// TIA Portal V19 export
FUNCTION "FC_Niveau_St" : Void   // FC96, STL
TITLE = Badniveau-Steuerungen
{ S7_Optimized_Access := 'FALSE' }
AUTHOR : RE
NAME : FC_nass
VERSION : 2.0
// stored: AutoNumber false
   VAR_TEMP
      Freigabe : Bool;
   END_VAR
BEGIN

NETWORK
TITLE = Niveau-Regelungen/Nachspeisungen/Spritzregister
      CLR;
      =     "DB_NSP".Test_on;

      CALL  "FC_Nachspeisung";

      A     "DB_ANLAGE".BA.Simulation;
      BEC;


NETWORK
TITLE = CM01
      A     "Panel".CM01.NSP_Auto;
      =     "DB_Panel_Posinfo".Pos[1].NS_Auto;

// Becken leer und keine Dosierung aktiv
      AN    "DB_POS".POS[1].belegt;
      AN    "DB_POS".POS[2].belegt;
      AN    "DB_POS".POS[3].belegt;
      AN    "DB_POS".POS[4].belegt;
      AN    "DB_POS".POS[5].belegt;
      AN    "DB_POS".POS[6].belegt;
      AN    "DB_DP".DP[1].Dosi_akt;
      AN    "DB_DP".DP[2].Dosi_akt;
      AN    "DB_DP".DP[5].Dosi_akt;
      AN    "DB_DP".DP[6].Dosi_akt;
      =     "DB_NSP".NSP[1].Freigabe;

      A     "E_Niv_Min_CM01.BL03";
      =     "DB_NSP".NSP[1].Niveau_ok;
      =     "DB_NSP".NSP[2].Niveau_ok;
      =     "DB_NSP".NSP[3].Niveau_ok;
      =     "DB_NSP".NSP[4].Niveau_ok;
      =     "DB_NSP".NSP[5].Niveau_ok;
      =     "DB_NSP".NSP[6].Niveau_ok;
      NOT;
      =     "DB_NSP".NSP[1].AL_Niv_min;

// Dosierungen gegeneinander verriegeln
// Verwerfen hat Vorrang
      A     "DB_DP".DP[1].Dosi_akt;
      O     "DB_DP".DP[5].Dosi_akt;
      O     "DB_DP".DP[3].Dosi_akt;
      O     "DB_DP".DP[7].Dosi_akt;
      S     "DB_DP".DP[2].DP_OFF;
      S     "DB_DP".DP[6].DP_OFF;
      S     "DB_DP".DP[4].DP_OFF;
      S     "DB_DP".DP[8].DP_OFF;
      JC    Ents;

// CM01 gewinnt
      A     "DB_DP".DP[2].Dosi_akt;  //CM01
      O     "DB_DP".DP[6].Dosi_akt;
      A(;
      A     "DB_DP".DP[4].Dosi_akt;  //CM02
      O     "DB_DP".DP[8].Dosi_akt;
      );
      AN    "DB_DP".DP[2].DP_OFF;
      AN    "DB_DP".DP[6].DP_OFF;
      S     "DB_DP".DP[4].DP_OFF;
      S     "DB_DP".DP[8].DP_OFF;
      JC    Ents;

      A     "DB_DP".DP[2].Dosi_akt;  //CM01
      O     "DB_DP".DP[6].Dosi_akt;
      AN    "DB_DP".DP[2].DP_OFF;
      AN    "DB_DP".DP[6].DP_OFF;
      =     "DB_DP".DP[4].DP_OFF;
      =     "DB_DP".DP[8].DP_OFF;

      A     "DB_DP".DP[4].Dosi_akt;  //CM02
      O     "DB_DP".DP[8].Dosi_akt;
      AN    "DB_DP".DP[4].DP_OFF;
      AN    "DB_DP".DP[8].DP_OFF;
      =     "DB_DP".DP[2].DP_OFF;
      =     "DB_DP".DP[6].DP_OFF;

//Verwerfen - alles aus
Ents: AN    "DB_DP".DP[1].Dosi_akt;
      AN    "DB_DP".DP[3].Dosi_akt;
      AN    "DB_DP".DP[5].Dosi_akt;
      AN    "DB_DP".DP[7].Dosi_akt;
      R     "DB_DP".DP[1].DP_OFF;
      R     "DB_DP".DP[3].DP_OFF;
      R     "DB_DP".DP[5].DP_OFF;
      R     "DB_DP".DP[7].DP_OFF;

// Verwerfen CM01 gewinnt
      A     "DB_DP".DP[1].Dosi_akt;  //CM01
      O     "DB_DP".DP[5].Dosi_akt;
      A(;
      A     "DB_DP".DP[3].Dosi_akt;  //CM02
      O     "DB_DP".DP[7].Dosi_akt;
      );
      AN    "DB_DP".DP[1].DP_OFF;
      AN    "DB_DP".DP[5].DP_OFF;
      S     "DB_DP".DP[3].DP_OFF;
      S     "DB_DP".DP[7].DP_OFF;
      JC    CM01;

      A     "DB_DP".DP[1].Dosi_akt;  //CM01
      O     "DB_DP".DP[5].Dosi_akt;
      AN    "DB_DP".DP[1].DP_OFF;
      AN    "DB_DP".DP[5].DP_OFF;
      =     "DB_DP".DP[3].DP_OFF;
      =     "DB_DP".DP[7].DP_OFF;

      A     "DB_DP".DP[3].Dosi_akt;  //CM02
      O     "DB_DP".DP[7].Dosi_akt;
      AN    "DB_DP".DP[3].DP_OFF;
      AN    "DB_DP".DP[7].DP_OFF;
      =     "DB_DP".DP[1].DP_OFF;
      =     "DB_DP".DP[5].DP_OFF;

CM01: NOP   0;
// Anforderung bilden
// Nachschärfen
      A     "DB_NSP".NSP[1].Nachspeisen;
      O(;
      A     "DB_DP".DP[2].Dosi_akt;
      AN    "DB_DP".DP[2].DP_OFF;
      );
      O(;
      A     "DB_DP".DP[6].Dosi_akt;
      AN    "DB_DP".DP[6].DP_OFF;
      );
      A     "Pu_GP01.GP13".In.Auto;
      A     "Pu_GP01.GP13".Out.Versorgung_UV01;
      AN    "Pu_GP02.GP10".In.Anf_HF_CM01;
      =     "Pu_GP01.GP13".In.Anf_HF_CM01;

      A     "DB_NSP".NSP[1].Nachspeisen;
      O(;
      A     "DB_DP".DP[2].Dosi_akt;
      AN    "DB_DP".DP[2].DP_OFF;
      );
      O(;
      A     "DB_DP".DP[6].Dosi_akt;
      AN    "DB_DP".DP[6].DP_OFF;
      );
      A     "Pu_GP02.GP10".In.Auto;
      A     "Pu_GP02.GP10".Out.Versorgung_UV01;
      AN    "Pu_GP01.GP13".In.Anf_HF_CM01;
      =     "Pu_GP02.GP10".In.Anf_HF_CM01;

// Verwerfen
      A     "DB_DP".DP[1].Dosi_akt;
      AN    "DB_DP".DP[1].DP_OFF;
      O(;
      A     "DB_DP".DP[5].Dosi_akt;
      AN    "DB_DP".DP[5].DP_OFF;
      );
      A     "UP_CM01.GP02".In.Auto;
      A(;
      A     "UP_CM01.GP02".In."SRM_GP01.QM14_auf";
      O     "UP_CM01.GP02".In."SRM_GP02.QM41_auf";
      );
      =     "UP_CM01.GP02".In.Anf_HF_Ents_CM0x;

// WT-zählergesteuert (DP1/2)
      A     "Panel".CM01.Dosierung_LF;
      R     "DB_Panel_DP".DoPu[1].Auto;
      R     "DB_Panel_DP".DoPu[2].Auto;

// LF-gesteuert (DP(5/6)
      CALL  "ToDo";

      A     "DB_DP".DP[5].Dosi_akt;
      O     "DB_DP".DP[6].Dosi_akt;
      L     S5T#15m;
      SF    "TA-Pause_LF_CM01";

      AN    "Panel".CM01.Dosierung_LF;
      R     "DB_Panel_DP".DoPu[5].Auto;
      R     "DB_Panel_DP".DoPu[6].Auto;
      JC    LF1E;

      L     "Panel".IW."LF_CM01.BN02";
      L     "Panel".CM01.Sollwert_LF;
      <R;  // ???
      AN    "TA-Pause_LF_CM01";
      AN    "DB_DP".DP[5].AM_DP_Start;
      AN    "DB_DP".DP[6].AM_DP_Start;
      S     "DB_DP".DP[5].DP_Start;
      S     "DB_DP".DP[5].AM_DP_Start;
      S     "DB_DP".DP[6].DP_Start;
      S     "DB_DP".DP[6].AM_DP_Start;
      JC    LF1E;

      A     "DB_DP".DP[5].Dosi_akt;
      R     "DB_DP".DP[5].AM_DP_Start;

      A     "DB_DP".DP[6].Dosi_akt;
      R     "DB_DP".DP[6].AM_DP_Start;

LF1E: NOP   0;


NETWORK
TITLE = CM02
      A     "Panel".CM02.NSP_Auto;
      =     "DB_Panel_Posinfo".Pos[13].NS_Auto;

// Becken leer und keine Dosierung aktiv
      AN    "DB_POS".POS[13].belegt;
      AN    "DB_POS".POS[14].belegt;
      AN    "DB_POS".POS[15].belegt;
      AN    "DB_POS".POS[16].belegt;
      AN    "DB_POS".POS[17].belegt;
      AN    "DB_POS".POS[18].belegt;
      AN    "DB_DP".DP[3].Dosi_akt;
      AN    "DB_DP".DP[4].Dosi_akt;
      AN    "DB_DP".DP[7].Dosi_akt;
      AN    "DB_DP".DP[8].Dosi_akt;
      =     "DB_NSP".NSP[13].Freigabe;

      A     "E_Niv_Min_CM02.BL10";
      =     "DB_NSP".NSP[13].Niveau_ok;
      =     "DB_NSP".NSP[14].Niveau_ok;
      =     "DB_NSP".NSP[15].Niveau_ok;
      =     "DB_NSP".NSP[16].Niveau_ok;
      =     "DB_NSP".NSP[17].Niveau_ok;
      =     "DB_NSP".NSP[18].Niveau_ok;
      NOT;
      =     "DB_NSP".NSP[13].AL_Niv_min;


// Anforderung bilden
// Nachschärfen
      A     "DB_NSP".NSP[13].Nachspeisen;
      O(;
      A     "DB_DP".DP[4].Dosi_akt;
      AN    "DB_DP".DP[4].DP_OFF;
      );
      O(;
      A     "DB_DP".DP[8].Dosi_akt;
      AN    "DB_DP".DP[8].DP_OFF;
      );
      A     "Pu_GP01.GP13".In.Auto;
      A     "Pu_GP01.GP13".Out.Versorgung_UV01;
      AN    "Pu_GP02.GP10".In.Anf_HF_CM02;
      =     "Pu_GP01.GP13".In.Anf_HF_CM02;

      A     "DB_NSP".NSP[13].Nachspeisen;
      O(;
      A     "DB_DP".DP[4].Dosi_akt;
      AN    "DB_DP".DP[4].DP_OFF;
      );
      O(;
      A     "DB_DP".DP[8].Dosi_akt;
      AN    "DB_DP".DP[8].DP_OFF;
      );
      A     "Pu_GP02.GP10".In.Auto;
      A     "Pu_GP02.GP10".Out.Versorgung_UV01;
      AN    "Pu_GP01.GP13".In.Anf_HF_CM02;
      =     "Pu_GP02.GP10".In.Anf_HF_CM02;

// Verwerfen
      A     "DB_DP".DP[3].Dosi_akt;
      AN    "DB_DP".DP[3].DP_OFF;
      O(;
      A     "DB_DP".DP[7].Dosi_akt;
      AN    "DB_DP".DP[7].DP_OFF;
      );
      A     "UP_CM02.GP05".In.Auto;
      A(;
      A     "UP_CM02.GP05".In."SRM_GP01.QM14_auf";
      O     "UP_CM02.GP05".In."SRM_GP02.QM41_auf";
      );
      =     "UP_CM02.GP05".In.Anf_HF_Ents_CM0x;

// WT-zählergesteuert (DP3/4)
      A     "Panel".CM02.Dosierung_LF;
      R     "DB_Panel_DP".DoPu[3].Auto;
      R     "DB_Panel_DP".DoPu[4].Auto;

// LF-gesteuert (DP(7/8)
      CALL  "ToDo";

      A     "DB_DP".DP[7].Dosi_akt;
      O     "DB_DP".DP[8].Dosi_akt;
      L     S5T#15m;
      SF    "TA-Pause_LF_CM02";

      AN    "Panel".CM02.Dosierung_LF;
      R     "DB_Panel_DP".DoPu[7].Auto;
      R     "DB_Panel_DP".DoPu[8].Auto;
      JC    LF2E;

      L     "Panel".IW."LF_CM02.BN04";
      L     "Panel".CM02.Sollwert_LF;
      <R;  // ???
      AN    "TA-Pause_LF_CM02";
      AN    "DB_DP".DP[7].AM_DP_Start;
      AN    "DB_DP".DP[8].AM_DP_Start;
      S     "DB_DP".DP[7].DP_Start;
      S     "DB_DP".DP[7].AM_DP_Start;
      S     "DB_DP".DP[8].DP_Start;
      S     "DB_DP".DP[8].AM_DP_Start;
      JC    LF2E;

      A     "DB_DP".DP[7].Dosi_akt;
      R     "DB_DP".DP[7].AM_DP_Start;

      A     "DB_DP".DP[8].Dosi_akt;
      R     "DB_DP".DP[8].AM_DP_Start;

LF2E: NOP   0;


NETWORK
TITLE = CM03

      A     "Panel".CM03.SPR_Auto;
      =     "DB_Panel_Posinfo".Pos[7].SR_Auto;
      =     "DB_Panel_Posinfo".Pos[8].SR_Auto;
      =     "DB_Panel_Posinfo".Pos[9].SR_Auto;
      =     "DB_Panel_Posinfo".Pos[10].SR_Auto;
      =     "DB_Panel_Posinfo".Pos[11].SR_Auto;
      =     "DB_Panel_Posinfo".Pos[12].SR_Auto;

      A     "Panel".CM03.SPR_Start_Test;
      R     "Panel".CM03.SPR_Start_Test;
      JCN   ST03;
      L     "Panel".CM03.SPR_Zeit_Test;
      T     "DB_Panel_Posinfo".Pos[7].T_Zt_SR;

ST03: A     "Panel".CM03.SPR_Stopp_Test;
      R     "Panel".CM03.SPR_Stopp_Test;
      JCN   FN03;
      L     0;
      T     "DB_Panel_Posinfo".Pos[7].T_Zt_SR;

//Pos.7..12
FN03: AN    "T_VEW_niO";
      A     "E_Niv_Uel_CM05.BL12";
      =     "DB_NSP".NSP[7].Freigabe;
      =     "DB_NSP".NSP[8].Freigabe;
      =     "DB_NSP".NSP[9].Freigabe;
      =     "DB_NSP".NSP[10].Freigabe;
      =     "DB_NSP".NSP[11].Freigabe;
      =     "DB_NSP".NSP[12].Freigabe;

// Spritzregister: beim Heben und Senken
      A     "DB_NSP".NSP[7].Spritzen;
      O     "DB_NSP".NSP[8].Spritzen;
      O     "DB_NSP".NSP[9].Spritzen;
      O     "DB_NSP".NSP[10].Spritzen;
      O     "DB_NSP".NSP[11].Spritzen;
      O     "DB_NSP".NSP[12].Spritzen;
      AN    "T_VEW_niO";
      A     "E_Niv_Uel_CM05.BL12";
      =     "A_CM03.QM35";


NETWORK
TITLE = CM04
//Pos.19..24
      A     "Panel".CM04.SPR_Auto;
      =     "DB_Panel_Posinfo".Pos[19].SR_Auto;
      =     "DB_Panel_Posinfo".Pos[20].SR_Auto;
      =     "DB_Panel_Posinfo".Pos[21].SR_Auto;
      =     "DB_Panel_Posinfo".Pos[22].SR_Auto;
      =     "DB_Panel_Posinfo".Pos[23].SR_Auto;
      =     "DB_Panel_Posinfo".Pos[24].SR_Auto;

      A     "Panel".CM04.NSP_Auto;
      =     "DB_Panel_Posinfo".Pos[19].NS_Auto;
      =     "DB_Panel_Posinfo".Pos[20].NS_Auto;
      =     "DB_Panel_Posinfo".Pos[21].NS_Auto;
      =     "DB_Panel_Posinfo".Pos[22].NS_Auto;
      =     "DB_Panel_Posinfo".Pos[23].NS_Auto;
      =     "DB_Panel_Posinfo".Pos[24].NS_Auto;

      L     "Panel".CM04.NSP_Zeit;
      T     "DB_Panel_Posinfo".Pos[19].Zeit_NS;
      T     "DB_Panel_Posinfo".Pos[20].Zeit_NS;
      T     "DB_Panel_Posinfo".Pos[21].Zeit_NS;
      T     "DB_Panel_Posinfo".Pos[22].Zeit_NS;
      T     "DB_Panel_Posinfo".Pos[23].Zeit_NS;
      T     "DB_Panel_Posinfo".Pos[24].Zeit_NS;

      A     "Panel".CM04.SPR_Start_Test;
      R     "Panel".CM04.SPR_Start_Test;
      JCN   ST04;
      L     "Panel".CM04.SPR_Zeit_Test;
      T     "DB_Panel_Posinfo".Pos[19].T_Zt_SR;

ST04: A     "Panel".CM04.SPR_Stopp_Test;
      R     "Panel".CM04.SPR_Stopp_Test;
      JCN   NS04;
      L     0;
      T     "DB_Panel_Posinfo".Pos[19].T_Zt_SR;

NS04: A     "Panel".CM04.NSP_Start_Test;
      R     "Panel".CM04.NSP_Start_Test;
      JCN   SN04;
      L     "Panel".CM04.NSP_Zeit_Tes;
      T     "DB_Panel_Posinfo".Pos[19].T_Zt_NS;

SN04: A     "Panel".CM04.NSP_Stopp_Test;
      R     "Panel".CM04.NSP_Stopp_Test;
      JCN   FN04;
      L     0;
      T     "DB_Panel_Posinfo".Pos[19].T_Zt_NS;

FN04: AN    "T_VEW_niO";
      A     "E_Niv_Uel_CM05.BL12";
      =     "DB_NSP".NSP[19].Freigabe;
      =     "DB_NSP".NSP[20].Freigabe;
      =     "DB_NSP".NSP[21].Freigabe;
      =     "DB_NSP".NSP[22].Freigabe;
      =     "DB_NSP".NSP[23].Freigabe;
      =     "DB_NSP".NSP[24].Freigabe;

// Spritzregister: beim Heben
      A     "DB_NSP".NSP[19].Spritzen;
      O     "DB_NSP".NSP[20].Spritzen;
      O     "DB_NSP".NSP[21].Spritzen;
      O     "DB_NSP".NSP[22].Spritzen;
      O     "DB_NSP".NSP[23].Spritzen;
      O     "DB_NSP".NSP[24].Spritzen;
      AN    "T_VEW_niO";
      A     "E_Niv_Uel_CM05.BL12";
      =     "A_CM04.QM74";

// Nachspeisung
// Zeit pro Korb
// niveaugesteuert, wenn CM03 nicht belegt und "min"-Niveau nicht erreicht

      A     "E_Niv_Min_CM03.BL06";
      O     "DB_POS".POS[7].belegt;
      O     "DB_POS".POS[8].belegt;
      O     "DB_POS".POS[9].belegt;
      O     "DB_POS".POS[10].belegt;
      O     "DB_POS".POS[11].belegt;
      O     "DB_POS".POS[12].belegt;
      O     "A_CM04.QM74";
      =     "DB_NSP".NSP[19].Niveau_ok;
      =     "DB_NSP".NSP[20].Niveau_ok;
      =     "DB_NSP".NSP[21].Niveau_ok;
      =     "DB_NSP".NSP[22].Niveau_ok;
      =     "DB_NSP".NSP[23].Niveau_ok;
      =     "DB_NSP".NSP[24].Niveau_ok;
      NOT;  // Nicht Spritzen und Nachspeisen gleichzeitig
      =     "DB_NSP".NSP[19].AL_Niv_min;

// Nicht Spritzen und Nachspeisen gleichzeitig
      A     "DB_POS".POS[19].FW_Hebt;
      =     "DB_NSP".NSP[19].Warte_NSPT;
      A     "DB_POS".POS[20].FW_Hebt;
      =     "DB_NSP".NSP[20].Warte_NSPT;
      A     "DB_POS".POS[21].FW_Hebt;
      =     "DB_NSP".NSP[21].Warte_NSPT;
      A     "DB_POS".POS[22].FW_Hebt;
      =     "DB_NSP".NSP[22].Warte_NSPT;
      A     "DB_POS".POS[23].FW_Hebt;
      =     "DB_NSP".NSP[23].Warte_NSPT;
      A     "DB_POS".POS[24].FW_Hebt;
      =     "DB_NSP".NSP[24].Warte_NSPT;

      A     "DB_NSP".NSP[19].Nachspeisen;
      O     "DB_NSP".NSP[20].Nachspeisen;
      O     "DB_NSP".NSP[21].Nachspeisen;
      O     "DB_NSP".NSP[22].Nachspeisen;
      O     "DB_NSP".NSP[23].Nachspeisen;
      O     "DB_NSP".NSP[24].Nachspeisen;
      =     "A_CM04.QM77";

END_FUNCTION
